FUNCTION_BLOCK Q_FillAttributes (* Command change fill attributes ( Part 6 - F.32 ) *)
  (* Standard: ISO 11783-6; Description: This command is used to change the fill attributes in a fill attributes object. Return values iso_s16 - E_NO_ERR - OK - E_OVERFLOW - buffer overflow - E_NOACT - Command not possible in current state - E_NO_INSTANCE - No VT client available *)
  (* Version 1.0, 2022-07-08, franz *)
  (* Documentation:
  This command is used to change the fill attributes in a fill attributes object.
   Return values
   iso_s16
    - E_NO_ERR - OK
   - E_OVERFLOW - buffer overflow
   - E_NOACT - Command not possible in current state
   - E_NO_INSTANCE - No VT client available
  *)
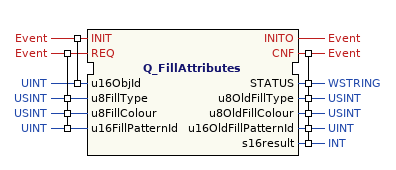
  EVENT_INPUT
    INIT WITH u16ObjId; (* Service Initialization *)
    REQ WITH u8FillType, u8FillColour, u16FillPatternId; (* Service Request *)
  END_EVENT
  EVENT_OUTPUT
    INITO; (* Initialization Confirm *)
    CNF WITH STATUS, u16OldFillPatternId, u8OldFillType, u8OldFillColour, s16result; (* Confirmation of Requested Service *)
  END_EVENT
  VAR_INPUT
    u16ObjId : UINT; (* Object ID *)
    u8FillType : USINT; (* New fill type (see Part 6 - B.14.4) *)
    u8FillColour : USINT; (* New fill colour (see Part 6 - B.14.4) *)
    u16FillPatternId : UINT; (* New fill pattern (see Part 6 - B.14.4) *)
  END_VAR
  VAR_OUTPUT
    STATUS : WSTRING; (* Service Status *)
    u8OldFillType : USINT; (* Old fill type (see Part 6 - B.14.4) *)
    u8OldFillColour : USINT; (* Old fill colour (see Part 6 - B.14.4) *)
    u16OldFillPatternId : UINT; (* Old fill pattern (see Part 6 - B.14.4) *)
    s16result : INT; (* retval see description *)
  END_VAR
END_FUNCTION_BLOCK
